Fanuc KAREL source: libind_pkt.kl

-- Software License Agreement (BSD License)
--
-- Copyright (c) 2012, 2013, TU Delft Robotics Institute
-- All rights reserved.
--
-- Redistribution and use in source and binary forms, with or without
-- modification, are permitted provided that the following conditions
-- are met:
--
--  * Redistributions of source code must retain the above copyright
--    notice, this list of conditions and the following disclaimer.
--  * Redistributions in binary form must reproduce the above
--    copyright notice, this list of conditions and the following
--    disclaimer in the documentation and/or other materials provided
--    with the distribution.
--  * Neither the name of the TU Delft Robotics Institute nor the names
--    of its contributors may be used to endorse or promote products
--    derived from this software without specific prior written
--    permission.
--
-- THIS SOFTWARE IS PROVIDED BY THE COPYRIGHT HOLDERS AND CONTRIBUTORS
-- "AS IS" AND ANY EXPRESS OR IMPLIED WARRANTIES, INCLUDING, BUT NOT
-- LIMITED TO, THE IMPLIED WARRANTIES OF MERCHANTABILITY AND FITNESS
-- FOR A PARTICULAR PURPOSE ARE DISCLAIMED. IN NO EVENT SHALL THE
-- COPYRIGHT OWNER OR CONTRIBUTORS BE LIABLE FOR ANY DIRECT, INDIRECT,
-- INCIDENTAL, SPECIAL, EXEMPLARY, OR CONSEQUENTIAL DAMAGES (INCLUDING,
-- BUT NOT LIMITED TO, PROCUREMENT OF SUBSTITUTE GOODS OR SERVICES;
-- LOSS OF USE, DATA, OR PROFITS; OR BUSINESS INTERRUPTION) HOWEVER
-- CAUSED AND ON ANY THEORY OF LIABILITY, WHETHER IN CONTRACT, STRICT
-- LIABILITY, OR TORT (INCLUDING NEGLIGENCE OR OTHERWISE) ARISING IN
-- ANY WAY OUT OF THE USE OF THIS SOFTWARE, EVEN IF ADVISED OF THE
-- POSSIBILITY OF SUCH DAMAGE.


PROGRAM libind_pkt
--------------------------------------------------------------------------------
--
-- Library routines for creating / processing ROS-Industrial packets
--
-- Note: in its current state this library can only deserialise
--       JOINT_POSITION (or JOINT) and JOINT_TRAJ_PT messages.
--
-- TODO: handle other types of incoming messages properly.
--
--
-- author: G.A. vd. Hoorn (TU Delft Robotics Institute)
--
--------------------------------------------------------------------------------
%NOLOCKGROUP
%NOPAUSE= COMMAND + TPENABLE + ERROR
%COMMENT = 'MFr15'




--------------------------------------------------------------------------------
--
-- local types & constants
--
--------------------------------------------------------------------------------
%INCLUDE include\libind_pkt_t
%INCLUDE include\ktype_sz_t




--------------------------------------------------------------------------------
--
-- remote routine prototypes
--
--------------------------------------------------------------------------------




--------------------------------------------------------------------------------
--
-- local routine prototypes
--
--------------------------------------------------------------------------------
%INCLUDE include\libind_pkt_h




--------------------------------------------------------------------------------
--
-- Empty body
--
--------------------------------------------------------------------------------
BEGIN
END libind_pkt




ROUTINE ipkt_ctor
BEGIN
	-- just reset packet
	ipkt_reset(this)
	-- cannot fail
	RETURN (0)
END ipkt_ctor




ROUTINE ipkt_reset
VAR
	len__ : INTEGER
	d__   : INTEGER
BEGIN
	--
	len__ = ARRAY_LEN(this.joint_data_)
	d__   = 0

	-- zero array with joint angles
	FOR d__ = 1 TO len__ DO
		this.joint_data_[d__] = 0.0
	ENDFOR
--
	---- set up ROS-Industrial packet fields
	--USING this DO
		---- default to JOINT_POSITION size
		--length_     = (RI_SZB_JPOS)
		--msg_type_   =  0
		--comm_type_  =  0
		--reply_type_ =  0
		--seq_nr_     =  0
		--duration_   =  0.0
		--velocity_   =  0.0
	--ENDUSING
END ipkt_reset




ROUTINE ipkt_srlise
VAR
	i__        : INTEGER
	stat__     : INTEGER
	array_sz__ : INTEGER
BEGIN
	-- .. and end with a CR
	WRITE fd(1) -- ACKNOWLEDGEMENT (4byte)
	WRITE fd(CR)

	-- done
	stat__ = IO_STATUS(fd)
	RETURN (-stat__)
END ipkt_srlise




ROUTINE ipkt_dsrlse
VAR
	i__        : INTEGER
	stat__     : INTEGER
	array_sz__ : INTEGER
BEGIN
	--
	i__ = 0
	stat__ = 0
	array_sz__ = 6 --ARRAY_LEN(this.joint_data_)


	-- now the array
	FOR i__ = 1 TO array_sz__ DO
		READ fd(this.joint_data_[i__])

		-- check
		stat__ = IO_STATUS(fd)
		IF stat__ <> 0 THEN RETURN (-stat__); ENDIF
	ENDFOR

	-- read footer. (dummy)
	READ fd(i__)
	stat__ = IO_STATUS(fd)
	IF stat__ <> 0 THEN RETURN (-stat__); ENDIF

	RETURN (-stat__)
END ipkt_dsrlse



ROUTINE ipkt_checkfd
VAR
	i__        : INTEGER
	stat__      : INTEGER
	bytes_ahd__ : INTEGER
BEGIN

	bytes_ahd__ = 0
	stat__      = 0


	WRITE TPDISPLAY('         ROUTINE ipkt_checkfd', CR)
	BYTES_AHEAD(fd, bytes_ahd__, stat__)
	WRITE TPDISPLAY('         BYTES_AHEAD(fd, bytes_ahd__, stat__)', CR)
	IF stat__ <> 0 THEN RETURN (-stat__); ENDIF

	-- is there enough for a packet?
	IF (bytes_ahd__ >= 30) THEN
		WRITE TPDISPLAY('         IF (bytes_ahd__  >= 30) THEN', CR)

		-- deserialise
		stat__ = ipkt_dsrlse(pkt, fd)
		WRITE TPDISPLAY('         stat__ = ipkt_dsrlse(pkt, fd)', CR)


		IF stat__ <> 0 THEN RETURN (-ABS(stat__)); ENDIF

		-- notify user of packet we deserialised
		RETURN (1)
	--
	ENDIF

	-- done
	RETURN (-ABS(stat__))

END ipkt_checkfd
